FUNCTION_BLOCK AGENT_GATE (* Diagnostic agent gateway Service Interface Function Block *)
  (* Standard: 61499-2; Description: Switchable gateway for passthrough of data that can be blocked and re-routed under control of the Fault Diagnostic Engine agents. *)
  (* Version 1.0, 2020-02-24, Badger, AUT *)
  (* Compiler header: #include <iostream> #include <stdio.h> #include "NIOclient.h" *)
  (* Compiler Other C++ C++ 1.0 *)
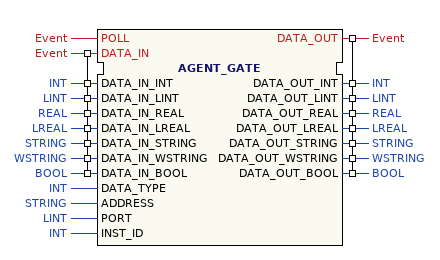
  EVENT_INPUT
    POLL; (* Poll the server to either switch the gate or get a data value. *)
    DATA_IN WITH DATA_IN_INT, DATA_IN_LINT, DATA_IN_REAL, DATA_IN_LREAL, DATA_IN_STRING, DATA_IN_WSTRING, DATA_IN_BOOL; (* Data in event *)
  END_EVENT
  EVENT_OUTPUT
    DATA_OUT WITH DATA_OUT_INT, DATA_OUT_LINT, DATA_OUT_REAL, DATA_OUT_LREAL, DATA_OUT_STRING, DATA_OUT_WSTRING, DATA_OUT_BOOL; (* Data out event *)
  END_EVENT
  VAR_INPUT
    DATA_IN_INT : INT;
    DATA_IN_LINT : LINT;
    DATA_IN_REAL : REAL;
    DATA_IN_LREAL : LREAL;
    DATA_IN_STRING : STRING;
    DATA_IN_WSTRING : WSTRING;
    DATA_IN_BOOL : BOOL;
    DATA_TYPE : INT;
    ADDRESS : STRING;
    PORT : LINT;
    INST_ID : INT;
  END_VAR
  VAR_OUTPUT
    DATA_OUT_INT : INT;
    DATA_OUT_LINT : LINT;
    DATA_OUT_REAL : REAL;
    DATA_OUT_LREAL : LREAL;
    DATA_OUT_STRING : STRING;
    DATA_OUT_WSTRING : WSTRING;
    DATA_OUT_BOOL : BOOL;
  END_VAR
  SERVICE APPLICATION/RESOURCE (* Diagnostic agent gateway Service Interface Function Block *)
    SEQUENCE normal_establishment
      APPLICATION.INIT+(PARAMS) -> RESOURCE.initialize(PARAMS) -> APPLICATION.INITO+();
    END_SEQUENCE
    SEQUENCE unsuccessful_establishment
      APPLICATION.INIT+(PARAMS) -> RESOURCE.initialize(PARAMS) -> APPLICATION.INITO-(STATUS);
    END_SEQUENCE
    SEQUENCE request_confirm
      APPLICATION.REQ+(SD) -> RESOURCE.request(SD) -> APPLICATION.CNF+(RD);
    END_SEQUENCE
    SEQUENCE request_inhibited
      APPLICATION.REQ-(SD) -> APPLICATION.CNF-(STATUS);
    END_SEQUENCE
    SEQUENCE request_error
      APPLICATION.REQ+(SD) -> RESOURCE.request(SD) -> APPLICATION.CNF-(STATUS);
    END_SEQUENCE
    SEQUENCE indication_response
      RESOURCE.indicate(RD) -> APPLICATION.IND+(RD);
      APPLICATION.RSP(QI,SD) -> RESOURCE.response(QI,SD);
    END_SEQUENCE
    SEQUENCE indication_inhibited
      RESOURCE.indicate(RD,QI=FALSE) -> RESOURCE.inhibited();
    END_SEQUENCE
    SEQUENCE error_indication
      RESOURCE.error(STATUS) -> APPLICATION.IND-(STATUS);
    END_SEQUENCE
    SEQUENCE application_initiated_termination
      APPLICATION.INIT-() -> RESOURCE.terminate() -> APPLICATION.INITO-(STATUS);
    END_SEQUENCE
    SEQUENCE resource_initiated_termination
      -> APPLICATION.INITO-(STATUS);
    END_SEQUENCE
  END_SERVICE
END_FUNCTION_BLOCK
